{attribute 'TcGenerated'}
{attribute 'no-analysis'}
{attribute 'linkalways'}
// This function has been automatically generated from the project information.
VAR_GLOBAL CONSTANT
    {attribute 'const_non_replaced'}
    stLibVersion_TcoPneumatics : ST_LibVersion := (
        iMajor := 0,
        iMinor := 1,
        iBuild := 0,
        iRevision := 54,
        nFlags := 0,
        sVersion := '0.1.0.54');
END_VAR

(* stored: Version 1.1.0.1, ProductVersion 3.1.4024.6
   GVL Global_Version: Id {d36f533e-f5f4-4932-9782-ef6481cd4e92} *)
